// TwinCAT 3 PLC project PyADSTest
// ProgramVersion: 3.1.4024.0
// libraries:
//   Tc2_Standard, * (Beckhoff Automation GmbH)
//   Tc2_System, * (Beckhoff Automation GmbH)
//   Tc3_Module, * (Beckhoff Automation GmbH)
// project tree:
//   DUTs/ stStruct.TcDUT
//   GVLs/ Globals.TcGVL
//   / PlcTask.TcTTO
//   POUs/ MAIN.TcPOU
// real-time tasks:
//   TASK PlcTask: cycle T#10ms, priority 20, ADS port 350

CONFIGURATION PyADSTest
    RESOURCE PLC ON TwinCAT3
        TASK PlcTask(INTERVAL := T#10ms, PRIORITY := 20);
        PROGRAM MAIN WITH PlcTask : MAIN;
    END_RESOURCE
END_CONFIGURATION

// ---- DUTs/stStruct.TcDUT
TYPE stStruct :
STRUCT
	bFirst : BOOL;
	iSecond : INT;
	rThird : REAL;	
END_STRUCT
END_TYPE

// ---- GVLs/Globals.TcGVL
{attribute 'qualified_only'}
VAR_GLOBAL
	bBool1 : BOOL := FALSE;
	bBool2 : BOOL := TRUE;
END_VAR

// ---- POUs/MAIN.TcPOU
PROGRAM MAIN
VAR
	bOut1 : BOOL;
	bOut2 : BOOL;
	iNumber : INT := 50;
	stStruct : stStruct;
END_VAR

bOut1 := Globals.bBool1;
bOut2 := Globals.bBool2;
stStruct.bFirst := TRUE;
stStruct.iSecond := 5;
stStruct.rThird := 1.3;

END_PROGRAM
